// TIA Portal V18 export
// export: Created 2026-06-09T02:47:52.7180682Z, ExportSetting WithDefaults, DisplayName Totally Integrated Automation Portal, DisplayVersion V18, DisplayName TIA Portal Openness, DisplayVersion V18, DisplayName TIA Portal Version Control Interface, DisplayVersion V18, DisplayName STEP 7 Professional, DisplayVersion V18, DisplayName STEP 7 Safety, DisplayVersion V18, DisplayName WinCC Professional, DisplayVersion V18
ORGANIZATION_BLOCK "Main"   // OB1, LAD, ProgramCycle
TITLE = "Main Program Sweep (Cycle)"
{ S7_Optimized_Access := 'TRUE' }
VERSION : 0.1
// stored: AutoNumber true, IsIECCheckEnabled false, SetENOAutomatically false
   VAR_INPUT
      Initial_Call : Bool;   // Initial call of this OB
      Remanence : Bool;   // =True, if remanent data are available
   END_VAR
   VAR_TEMP   // added for the SCL form of the ladder/FBD networks
      _w1 : Bool;
      _w2 : Bool;
      _w3 : Bool;
      _w4 : Bool;
      _w5 : Bool;
   END_VAR
BEGIN

REGION Network 1
   // Linię produkcyjną uruchamiamy poprzez włącznik główny oraz dodatkowo każdy etap produkcji na panelu HMI.
   // Wyłącznik bezpieczeństwa znajduje się w kilku miejscach na linii produkcyjnej.
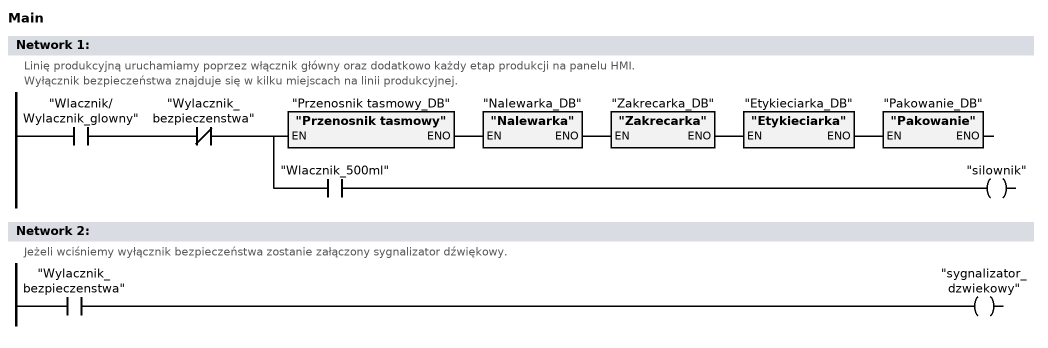
   RUNG wire#powerrail
      Contact( "Wlacznik/Wylacznik_glowny" )
      I_Contact( "Wylacznik_bezpieczenstwa" )
      wire#w1
      "Przenosnik tasmowy_DB"()
      "Nalewarka_DB"()
      "Zakrecarka_DB"()
      "Etykieciarka_DB"()
      "Pakowanie_DB"()
   END_RUNG
   RUNG wire#w1
      Contact( "Wlacznik_500ml" )
      Coil( "silownik" )
   END_RUNG
   // the same network as SCL:
   #_w1 := "Wlacznik/Wylacznik_glowny" AND NOT "Wylacznik_bezpieczenstwa";
   "Przenosnik tasmowy_DB"(EN := #_w1, ENO => #_w2);   // "Przenosnik tasmowy"
   "Nalewarka_DB"(EN := #_w2, ENO => #_w3);   // "Nalewarka"
   "Zakrecarka_DB"(EN := #_w3, ENO => #_w4);   // "Zakrecarka"
   "Etykieciarka_DB"(EN := #_w4, ENO => #_w5);   // "Etykieciarka"
   IF #_w5 THEN
       "Pakowanie_DB"();   // "Pakowanie"
   END_IF;
   "silownik" := #_w1 AND "Wlacznik_500ml";
END_REGION

REGION Network 2
   // Jeżeli wciśniemy wyłącznik bezpieczeństwa zostanie załączony sygnalizator dźwiękowy.
   RUNG wire#powerrail
      Contact( "Wylacznik_bezpieczenstwa" )
      Coil( "sygnalizator_dzwiekowy" )
   END_RUNG
   // the same network as SCL:
   "sygnalizator_dzwiekowy" := "Wylacznik_bezpieczenstwa";
END_REGION
END_ORGANIZATION_BLOCK
